{attribute 'conditionalshow'}
TYPE ST_ProfidriveParam :
STRUCT
	nAttribute	: BYTE;
	nNumber		: UINT;
	nSubIndex	: UINT;
	nElements	: BYTE;
	nFormat		: E_ProfidriveParamFormat;
	aValue		: ARRAY[0..234] OF BYTE;
END_STRUCT
END_TYPE

(* stored: Version 1.1.0.1, ProductVersion 3.1.4024.12
   DUT ST_ProfidriveParam: Id {f5776013-df66-0140-29e6-8017663fcb6a} *)
